FUNCTION_BLOCK Pure
  (* Version 1.0, 2007-10-25, Goran Cengic, Chalmers *)
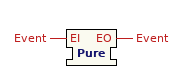
  EVENT_INPUT
    EI;
  END_EVENT
  EVENT_OUTPUT
    EO;
  END_EVENT
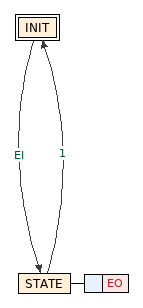
  EC_STATES
    INIT;
    STATE : -> EO;
  END_STATES
  EC_TRANSITIONS
    INIT TO STATE := EI;
    STATE TO INIT := 1;
  END_TRANSITIONS
END_FUNCTION_BLOCK
